FUNCTION_BLOCK LINEAR_MOVE (* Linear movement *)
  (* Standard: 61499-2 *)
  (* Version 1.0, 23-12-11, Guilherme Jarentchuk, Universidade do Estado de Santa Catarina *)
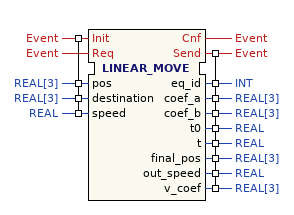
  EVENT_INPUT
    Init WITH pos, destination, speed; (* Initialization Request *)
    Req; (* Requisition to finish *)
  END_EVENT
  EVENT_OUTPUT
    Cnf; (* Execution confirmed *)
    Send WITH eq_id, coef_a, coef_b, t0, t, final_pos, out_speed, v_coef; (* Send data to output *)
  END_EVENT
  VAR_INPUT
    pos : ARRAY [0..2] OF REAL := [0,0,0]; (* Machine position *)
    destination : ARRAY [0..2] OF REAL; (* Destination point *)
    speed : REAL; (* Speed in m/s *)
  END_VAR
  VAR_OUTPUT
    eq_id : INT; (* Curve equation type id *)
    coef_a : ARRAY [0..2] OF REAL; (* Line angular coefficients *)
    coef_b : ARRAY [0..2] OF REAL; (* Line linear coefficients *)
    t0 : REAL; (* Initial parameter *)
    t : REAL; (* Final parameter *)
    final_pos : ARRAY [0..2] OF REAL; (* Final position *)
    out_speed : REAL; (* Speed in m/s *)
    v_coef : ARRAY [0..2] OF REAL; (* Velocity coefficients *)
  END_VAR
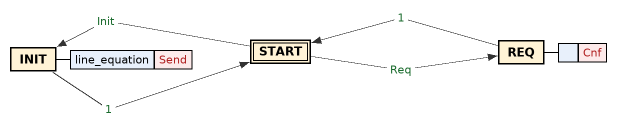
  EC_STATES
    START;
    REQ : -> Cnf;
    INIT : line_equation -> Send;
  END_STATES
  EC_TRANSITIONS
    START TO INIT := Init;
    START TO REQ := Req;
    REQ TO START := 1;
    INIT TO START := 1;
  END_TRANSITIONS
  ALGORITHM line_equation IN Lua:
 eq_id = 1 coef_a[1] = (destination[1] - pos[1]) coef_a[2] = (destination[2] - pos[2]) coef_a[3] = (destination[3] - pos[3]) coef_b[1] = pos[1] coef_b[2] = pos[2] coef_b[3] = pos[3] t0 = 0 t = 1 final_pos[1] = destination[1] final_pos[2] = destination[2] final_pos[3] = destination[3] out_speed = speed speed_mod = (coef_a[1]^2 + coef_a[2]^2 + coef_a[3]^2)^(0.5) v_coef[1] = coef_a[1]/speed_mod v_coef[2] = coef_a[2]/speed_mod v_coef[3] = coef_a[3]/speed_mod
  END_ALGORITHM
END_FUNCTION_BLOCK
